FUNCTION_BLOCK Helper (* Basic Function Block Type *)
  (* Standard: 61499-2 *)
  (* Version 0.0, 2010-11-22, 4DIAC-IDE, 4DIAC-Consortium *)
  (* Compiler header: package fb.rt.benchmarks; *)
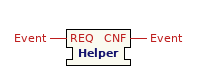
  EVENT_INPUT
    REQ; (* Normal Execution Request *)
  END_EVENT
  EVENT_OUTPUT
    CNF; (* Execution Confirmation *)
  END_EVENT
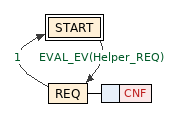
  EC_STATES
    START; (* Initial State *)
    REQ : -> CNF; (* Normal execution *)
  END_STATES
  EC_TRANSITIONS
    START TO REQ := EVAL_EV(Helper_REQ);
    REQ TO START := 1;
  END_TRANSITIONS
END_FUNCTION_BLOCK
